TYPE
    ST_PositionTable :
    STRUCT
        Zone  : STRING; // Object zone
        Index : INT; // The position index in the zone
        X_Pos : LREAL; // X-Axis target position (Unit: mm)
        Y_Pos : LREAL; // Y-Axis target position (Unit: mm)
        R_Pos : LREAL; // R-Axis target position (Unit: deg)
        Robot : INT; // unuse 
        Clip  : E_ClipNo; // Select Object clip no.
    END_STRUCT
END_TYPE

(* stored: Version 1.1.0.1, ProductVersion 3.1.4024.13
   DUT ST_PositionTable: Id {d60422c6-bd18-4133-9aa4-47af49762ca1} *)
